FUNCTION_BLOCK Product
  (* Version 1.0, 2007-08-28, Goran Cengic, Chalmers *)
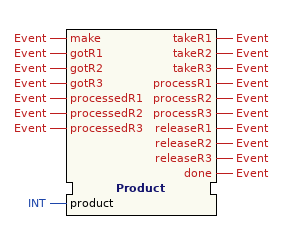
  EVENT_INPUT
    make;
    gotR1;
    gotR2;
    gotR3;
    processedR1;
    processedR2;
    processedR3;
  END_EVENT
  EVENT_OUTPUT
    takeR1;
    takeR2;
    takeR3;
    processR1;
    processR2;
    processR3;
    releaseR1;
    releaseR2;
    releaseR3;
    done;
  END_EVENT
  VAR_INPUT
    product : INT;
  END_VAR
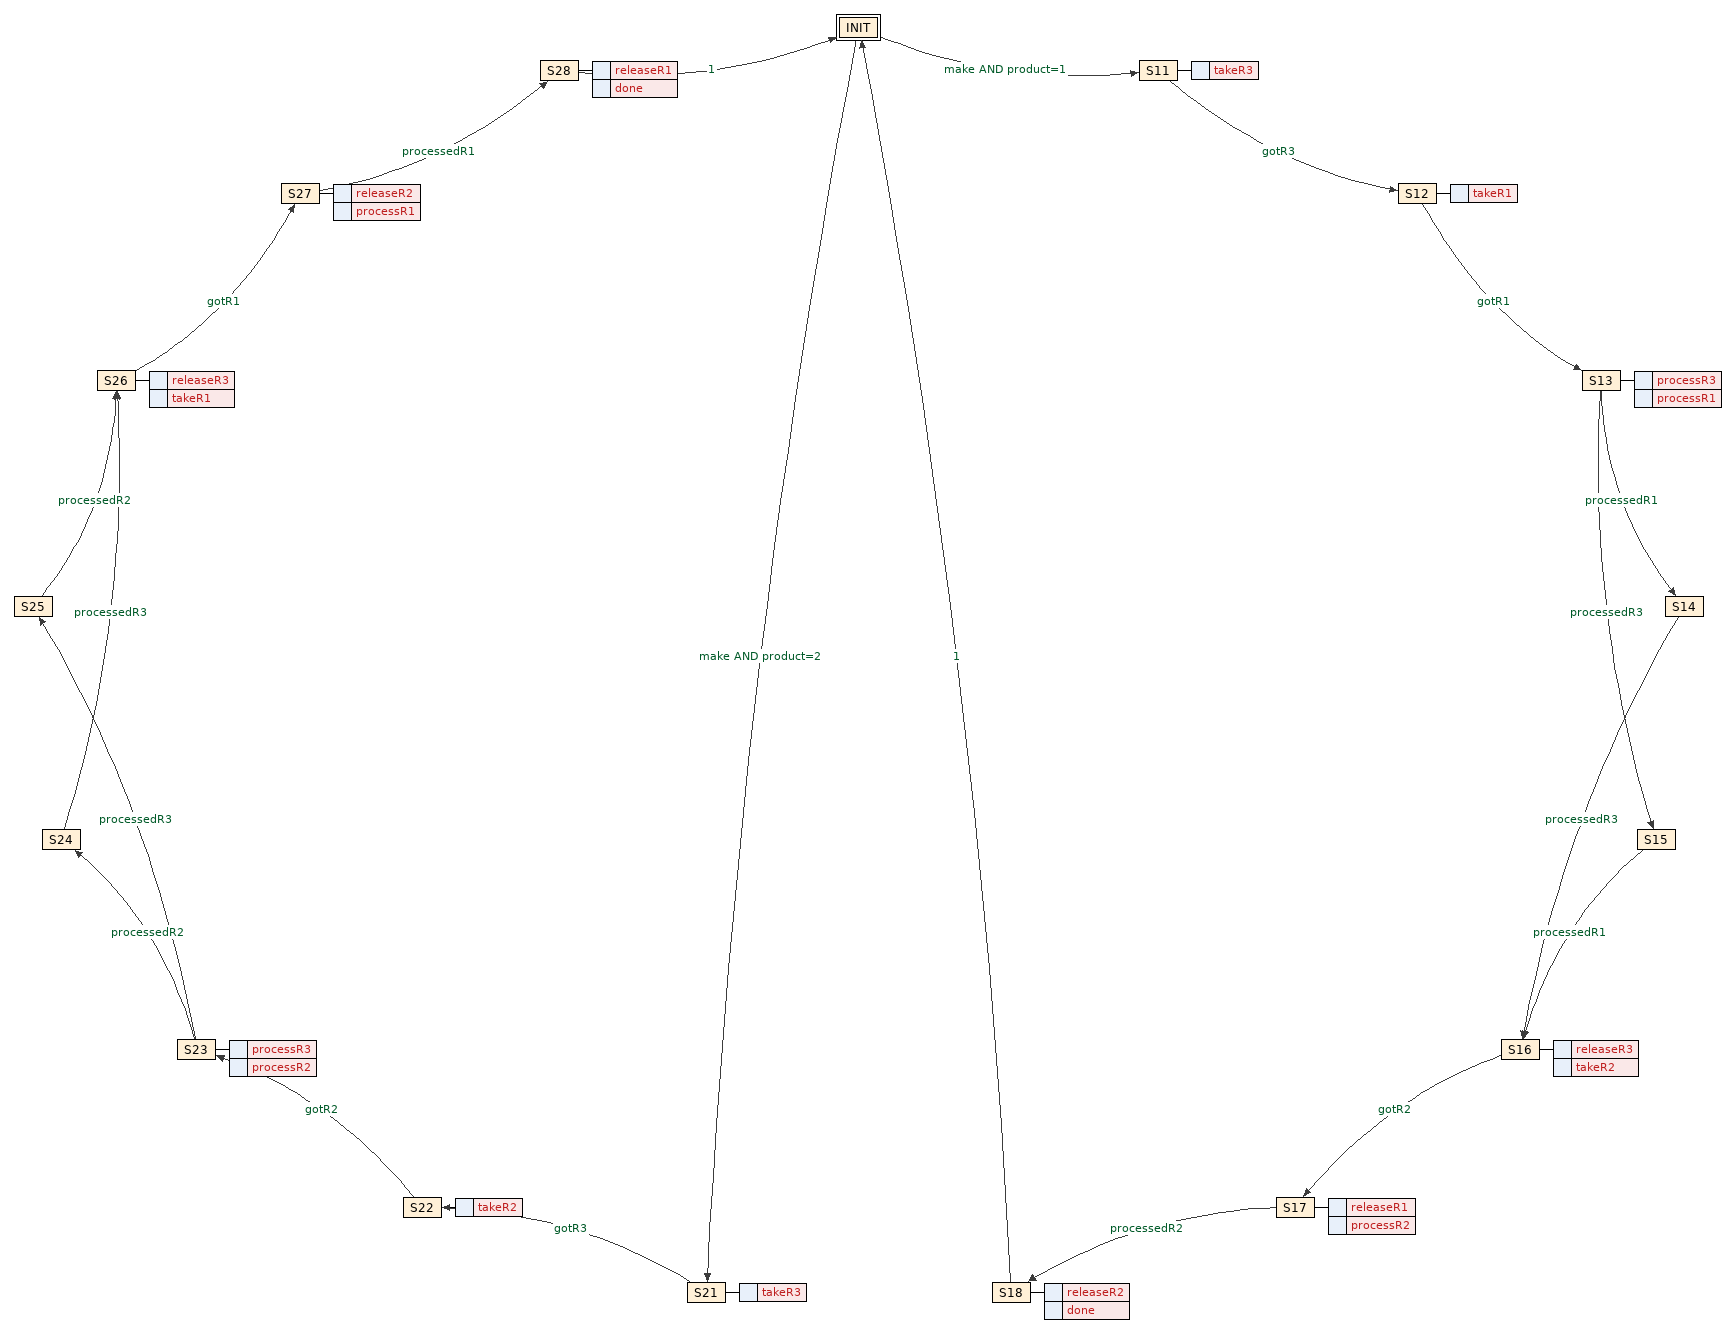
  EC_STATES
    INIT;
    S11 : -> takeR3;
    S12 : -> takeR1;
    S13 : -> processR3, -> processR1;
    S14;
    S15;
    S16 : -> releaseR3, -> takeR2;
    S17 : -> releaseR1, -> processR2;
    S18 : -> releaseR2, -> done;
    S21 : -> takeR3;
    S22 : -> takeR2;
    S23 : -> processR3, -> processR2;
    S24;
    S25;
    S26 : -> releaseR3, -> takeR1;
    S27 : -> releaseR2, -> processR1;
    S28 : -> releaseR1, -> done;
  END_STATES
  EC_TRANSITIONS
    INIT TO S11 := make AND product=1;
    S11 TO S12 := gotR3;
    S12 TO S13 := gotR1;
    S13 TO S14 := processedR1;
    S14 TO S16 := processedR3;
    S13 TO S15 := processedR3;
    S15 TO S16 := processedR1;
    S16 TO S17 := gotR2;
    S17 TO S18 := processedR2;
    S18 TO INIT := 1;
    INIT TO S21 := make AND product=2;
    S21 TO S22 := gotR3;
    S22 TO S23 := gotR2;
    S23 TO S24 := processedR2;
    S24 TO S26 := processedR3;
    S23 TO S25 := processedR3;
    S25 TO S26 := processedR2;
    S26 TO S27 := gotR1;
    S27 TO S28 := processedR1;
    S28 TO INIT := 1;
  END_TRANSITIONS
END_FUNCTION_BLOCK
